INTERFACE I_Receiver EXTENDS I_ReceiverNode, Tags.I_Tagged

METHOD Pair : Results.Result
VAR_INPUT
	iSignal		: I_Signal;
END_VAR
END_METHOD

METHOD Unpair : Results.Result
VAR_INPUT
	iSignal		: I_Signal;
END_VAR
END_METHOD

END_INTERFACE

(* stored: Version 1.1.0.1
   Itf I_Receiver: Id {e77ec887-f1b2-408f-a189-974b72e1bdf6}
   Method Pair: Id {838a7e8e-c8cf-40e5-97fc-565570b63c87}
   Method Unpair: Id {8cfd3959-a31b-46c5-b585-1cf014a69b98} *)
